(* CoDeSys 2.3.9.41 project: qqq1.pro *)
(* Libraries: Util.lib 18.5.10 15:14:28, STANDARD.LIB 4.10.05 11:14:46, IECSFC.LIB 13.4.06 15:51:28, ANALYZATION.LIB 5.10.99 09:05:06 *)

(* PLC configuration (modules and I/O channels)
Fast discrete inputs [I_SIMPLE_INPUT] node 0, in %IB0 out %QB0 {ChannellName = Fast discrete inputs; Filtrationtime = 10000}
  AT %IX0.0 [BitInput] Discrete input 1 {ChannellName = Enter name}
  AT %IX0.1 [BitInput] Discrete input 2 {ChannellName = Enter name}
z AT %IB1.0 [ByteInput] 8 discrete inputs {ChannellName = Enter name}
x AT %IB1.1 [ByteInput] 8 discrete inputs {ChannellName = Enter name}
Fast discrete outputs [OWEN_ID570] node 2, in %IB2 out %QB2 {ChannellName = Fast discrete outputs; SafeValueBool = FALSE; SafeValueBool = FALSE; SafeValueBool = FALSE; SafeValueBool = FALSE}
  AT %QX2.0 [BitOutput] Fast discrete output 1 {ChannellName = Enter name}
  AT %QX2.1 [BitOutput] Fast discrete output 2 {ChannellName = Enter name}
  AT %QX2.2 [BitOutput] Fast discrete output 3 {ChannellName = Enter name}
  AT %QX2.3 [BitOutput] Fast discrete output 4 {ChannellName = Enter name}
y AT %QB3.0 [ByteOutput] 8 discrete outputs {ChannellName = Enter name}
q AT %QB3.1 [ByteOutput] 8 discrete outputs {ChannellName = Enter name}
Special input [ID103] node 4, in %IB4 out %QB4 {ChannellName = Special input}
  AT %IX4.0 [BitInput] Special input {ChannellName = Enter name}
Special output [ID104] node 5, in %IB5 out %QB5 {ChannellName = Special output}
  AT %QX5.0 [BitOutput] Special output {ChannellName = Enter name}
TCP [TCP_ID221] node 1, in %IB6.0.1 out %QB6.0.1 {ChannellName = TCP; RemotePort = 502; Visibility = No}
RS-485-1 [COM1_USART] node 2, in %IB6.0.2 out %QB6.0.2 {ChannellName = RS-485-1; CommunicationSpeed = 115200; Parity = NO PARITY CHECK; BitLength = 8 bits; StopLength = One stop bit; InterfaceType = RS485; FrameOriented = RTU; Timeout = 0; Visibility = No}
in_tcp_1 AT %QB6.1.0 [ByteOutput] {ChannellName = Enter name}
tcp_out_1 AT %QB6.2.0 [ByteOutput] {ChannellName = Enter name}
count AT %QW6.3.0 [WordOutput] {ChannellName = Enter name}
ust AT %QW6.4.0 [WordOutput] {ChannellName = Enter name}
clk AT %QW6.5.0 [WordOutput] {ChannellName = Enter name}
*)

(* POU PLC_PRG, LD *)
PROGRAM PLC_PRG
VAR
	qqq: CTU;
	rr: WORD;
	BLINK: AnalyzeExpression;
	bbb: BLINK;
	e: BOOL;
	on_off: BOOL;
	reset: BOOL;
	rrr: CTU;
END_VAR
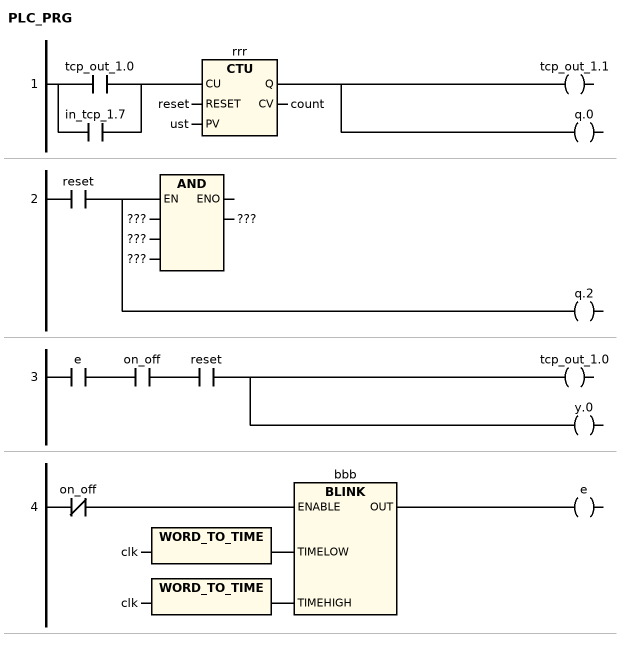
_LD_ (* Ladder Diagram *)
NETWORK 1
	{ [tcp_out_1.0] | [in_tcp_1.7] } - rrr:CTU(CU: *, RESET: reset, PV: ust, CV => count) --- (tcp_out_1.1) (q.0)
NETWORK 2
	[reset] --- (q.2)
		EN --- AND(???, ???, ???) => ???
NETWORK 3
	[e] - [on_off] - [reset] --- (tcp_out_1.0) (y.0)
NETWORK 4
	[/on_off] - bbb:BLINK(ENABLE: *, TIMELOW: WORD_TO_TIME(clk), TIMEHIGH: WORD_TO_TIME(clk)) --- (e)
_END_LD_
(* the same logic as Structured Text *)
(* Network 1 *)
rrr(CU := tcp_out_1.0 OR in_tcp_1.7, RESET := reset, PV := ust);
count := rrr.CV;
tcp_out_1.1 := rrr.Q;
q.0 := rrr.Q;
(* Network 2: see the listing above *)
(* Network 3 *)
tcp_out_1.0 := e AND on_off AND reset;
y.0 := tcp_out_1.0;
(* Network 4 *)
bbb(ENABLE := NOT on_off, TIMELOW := WORD_TO_TIME(clk), TIMEHIGH := WORD_TO_TIME(clk));
e := bbb.OUT;
END_PROGRAM

(* Visualisation tttr
rectangle at (60,30)-(161,111): invisible if .C
*)
